TYPE ST_ConveyorStatus :
STRUCT
    eState          : E_MachineState;

    bMotorRunning   : BOOL;

    bEntrySensor    : BOOL;
    bExitSensor     : BOOL;

    bFaultActive    : BOOL;

    nPartCount      : UDINT;
END_STRUCT
END_TYPE

(* stored: Version 1.1.0.1, ProductVersion 3.1.4026.18
   DUT ST_ConveyorStatus: Id {37e7da37-679a-46b0-9508-afde70681e6c} *)
